{library PUBLIC}
(* Position number type *)
TYPE PositionType : INT(1..9);
END_TYPE

(* stored: Version 1.1.0.1, ProductVersion 3.1.4022.12
   EnumerationTextList PositionType: Id {3b2b9b00-f006-40ee-9258-0307693aaba1} *)
